SUBAPPLICATION System_Tick (* Subapplication Type *)
  (* Standard: 61499-2 *)
  (* Version 1.0, 2026-08-07, franz *)
  PACKAGE MyLib::sys;
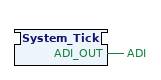
  PLUGS
    ADI_OUT : adapter::types::unidirectional::ADI;
  END_PLUGS
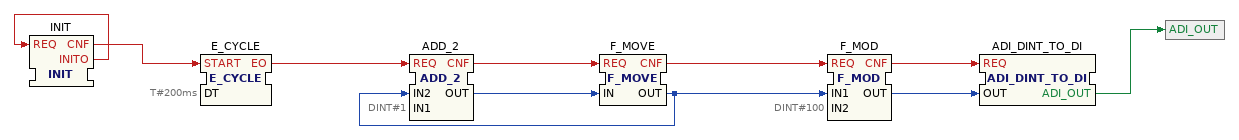
  FBS
    F_MOD : iec61131::arithmetic::F_MOD(IN2 := DINT#100);
    ADD_2 : iec61131::arithmetic::ADD_2(IN1 := DINT#1);
    E_CYCLE : iec61499::events::E_CYCLE(DT := T#200ms);
    INIT : iec61131::booleanOperators::INIT;
    F_MOVE : iec61131::selection::F_MOVE; {SET_ATTRIBUTE(DataType, DINT)}
    ADI_DINT_TO_DI : adapter::conversion::unidirectional::ADI_DINT_TO_DI;
  END_FBS
  EVENT_CONNECTIONS
    F_MOVE.CNF TO F_MOD.REQ;
    F_MOD.CNF TO ADI_DINT_TO_DI.REQ;
    E_CYCLE.EO TO ADD_2.REQ;
    ADD_2.CNF TO F_MOVE.REQ;
    INIT.CNF TO E_CYCLE.START;
    INIT.INITO TO INIT.REQ;
  END_CONNECTIONS
  DATA_CONNECTIONS
    F_MOVE.OUT TO F_MOD.IN1;
    F_MOD.OUT TO ADI_DINT_TO_DI.OUT;
    F_MOVE.OUT TO ADD_2.IN2;
    ADD_2.OUT TO F_MOVE.IN;
  END_CONNECTIONS
  ADAPTER_CONNECTIONS
    ADI_DINT_TO_DI.ADI_OUT TO ADI_OUT;
  END_CONNECTIONS
END_SUBAPPLICATION
